FUNCTION_BLOCK FB_MotorControl
VAR_INPUT
	AxisRef 	:	AXIS_REF;
	//Position
	//Ready
	//Reset
	
END_VAR
VAR_OUTPUT
		error	: BOOL;
END_VAR

(*Internals*)
VAR
	(* Properties *)
	Enabled : BOOL := FALSE;	


	eInitMotor : (START, IN_PROCESS, DONE, ERROR);	
	eMoveABS : (START, IN_PROCESS, DONE, ERROR);

	//stMC_Reset : ST_MC_Reset;
	

	stSA_Reset	:   ST_MC_Status;
	
	
	
	fbMcPower	:	MC_POWER;
	fbMcHome	: 	MC_HOME;
	fbMcJog		:	MC_JOG;
	
	// Global
	bError 		: BOOL	; // := TRUE;
	nErrorID 	: LINT	; //Check type
	
	//Reset
	fbMcReset	:	MC_RESET;
	fbTriggerReset : R_TRIG;
	bResetDone : BOOL := FALSE;
	
	
	
	fbMoveVelocity	: MC_MoveVelocity;
	fbMoveRelative	: MC_MoveRelative;
	fbMoveAbsolute	: MC_MoveAbsolute;
	
	fbHalt	: MC_Halt;
	fbStop	: MC_Stop;
	
	fbSA_GetPosition : MC_ReadActualPosition;
	
	//Input: Command
	bCmdResetExe			:	BOOL	;
	bCmdPowerEnable			:	BOOL	;
	bCmdPowerEnablePositive	:	BOOL	;
	bCmdPowerEnableNegative	:	BOOL	;
	bCmdHomeExecute			:	BOOL	;
	bSA_HomeCamInput	:	BOOL	;
	
	bSA_JogFwd			:	BOOL	;
	bSA_JogRev			:	BOOL	;
	
	bSA_HaltExe			: 	BOOL	;
	bSA_StopExe			: 	BOOL	;
	
	//stStatusMoveVelocity	: ST_MC_CMD	;
	stSA_VelCmd1	: ST_MC_CMD;
	stSA_RelCmd1			: ST_MC_CMD	;
	stSA_AbsCmd1			: ST_MC_CMD	;
	
	//Variables / Parameters
	lrSA_PowerOverride	: LREAL;
	lrSA_HomePosition	: LREAL;
	lrSA_SetPosition	: LREAL;
	lrSA_JogVelocity	: LREAL;
	
	//Status
	//stSA_Reset			: ST_MC_Status;
	stSA_Power			: ST_MC_Status;
	stSA_Home			: ST_MC_Status;
	stSA_SetPosition	: ST_MC_Status;
	stSA_Jog			: ST_MC_Status;
	stSA_GetPosition	: ST_MC_Status;
	
	
	stSA_VelSts1		: ST_MC_Status;
	stSA_MoveRelative		: ST_MC_Status;
	stSA_AbsSts1		: ST_MC_Status;
	
	stSA_Halt			: ST_MC_Status;
	stSA_Stop			: ST_MC_Status;

END_VAR

AxisRef.ReadStatus();
GetStatus();
//Here the state machine needs to be processed or farmed out.



//For a move

//Has position changed from the current target.....






//This should be removed as seperate methods are added.
ExecuteCommands();

PROPERTY bStateEnable : BOOL
GET
bStateEnable := Enabled ;
END_GET
SET
Enabled := bStateEnable;
END_SET
END_PROPERTY

METHOD PRIVATE Enable : BOOL
VAR_INPUT
END_VAR
END_METHOD

METHOD PRIVATE ExecuteCommands : BOOL
VAR_INPUT
END_VAR

VAR
END_VAR
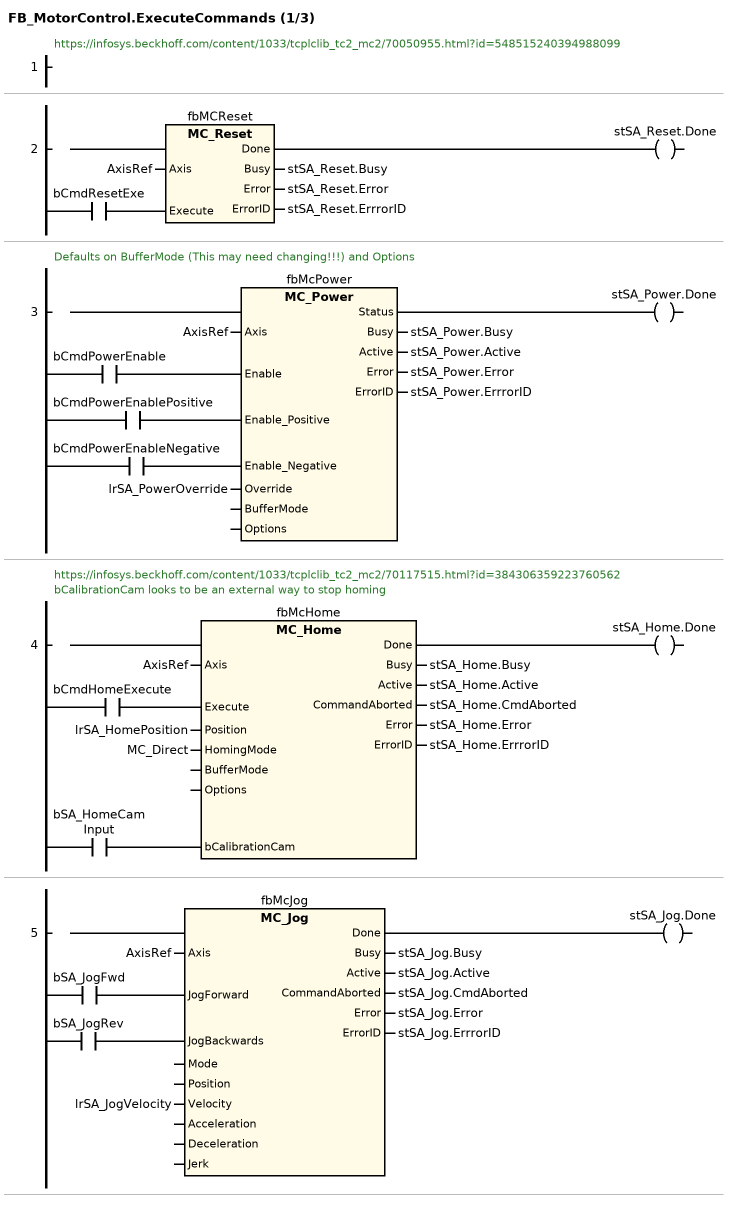
// NETWORK 1
// https://infosys.beckhoff.com/content/1033/tcplclib_tc2_mc2/70050955.html?id=548515240394988099

// NETWORK 2
fbMCReset(
    Axis := AxisRef,
    Execute := bCmdResetExe,
    Busy => stSA_Reset.Busy,
    Error => stSA_Reset.Error,
    ErrorID => stSA_Reset.ErrrorID); // MC_Reset
stSA_Reset.Done := fbMCReset.Done;

// NETWORK 3
// Defaults on BufferMode (This may need changing!!!) and Options
fbMcPower(
    Axis := AxisRef,
    Enable := bCmdPowerEnable,
    Enable_Positive := bCmdPowerEnablePositive,
    Enable_Negative := bCmdPowerEnableNegative,
    Override := lrSA_PowerOverride,
    Busy => stSA_Power.Busy,
    Active => stSA_Power.Active,
    Error => stSA_Power.Error,
    ErrorID => stSA_Power.ErrrorID); // MC_Power
stSA_Power.Done := fbMcPower.Status;

// NETWORK 4
// https://infosys.beckhoff.com/content/1033/tcplclib_tc2_mc2/70117515.html?id=384306359223760562
// bCalibrationCam looks to be an external way to stop homing
fbMcHome(
    Axis := AxisRef,
    Execute := bCmdHomeExecute,
    Position := lrSA_HomePosition,
    HomingMode := MC_Direct,
    bCalibrationCam := bSA_HomeCamInput,
    Busy => stSA_Home.Busy,
    Active => stSA_Home.Active,
    CommandAborted => stSA_Home.CmdAborted,
    Error => stSA_Home.Error,
    ErrorID => stSA_Home.ErrrorID); // MC_Home
stSA_Home.Done := fbMcHome.Done;

// NETWORK 5
fbMcJog(
    Axis := AxisRef,
    JogForward := bSA_JogFwd,
    JogBackwards := bSA_JogRev,
    Velocity := lrSA_JogVelocity,
    Busy => stSA_Jog.Busy,
    Active => stSA_Jog.Active,
    CommandAborted => stSA_Jog.CmdAborted,
    Error => stSA_Jog.Error,
    ErrorID => stSA_Jog.ErrrorID); // MC_Jog
stSA_Jog.Done := fbMcJog.Done;

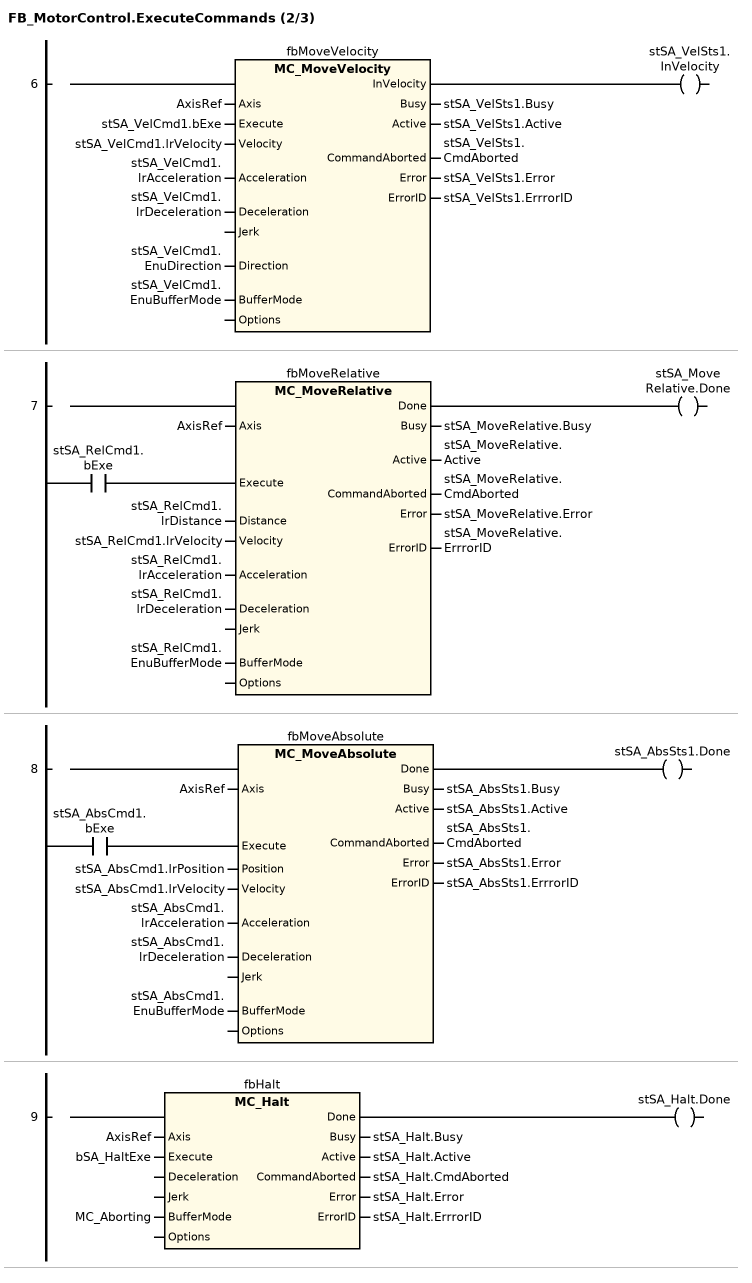
// NETWORK 6
fbMoveVelocity(
    Axis := AxisRef,
    Execute := stSA_VelCmd1.bExe,
    Velocity := stSA_VelCmd1.lrVelocity,
    Acceleration := stSA_VelCmd1.lrAcceleration,
    Deceleration := stSA_VelCmd1.lrDeceleration,
    Direction := stSA_VelCmd1.EnuDirection,
    BufferMode := stSA_VelCmd1.EnuBufferMode,
    Busy => stSA_VelSts1.Busy,
    Active => stSA_VelSts1.Active,
    CommandAborted => stSA_VelSts1.CmdAborted,
    Error => stSA_VelSts1.Error,
    ErrorID => stSA_VelSts1.ErrrorID); // MC_MoveVelocity
stSA_VelSts1.InVelocity := fbMoveVelocity.InVelocity;

// NETWORK 7
fbMoveRelative(
    Axis := AxisRef,
    Execute := stSA_RelCmd1.bExe,
    Distance := stSA_RelCmd1.lrDistance,
    Velocity := stSA_RelCmd1.lrVelocity,
    Acceleration := stSA_RelCmd1.lrAcceleration,
    Deceleration := stSA_RelCmd1.lrDeceleration,
    BufferMode := stSA_RelCmd1.EnuBufferMode,
    Busy => stSA_MoveRelative.Busy,
    Active => stSA_MoveRelative.Active,
    CommandAborted => stSA_MoveRelative.CmdAborted,
    Error => stSA_MoveRelative.Error,
    ErrorID => stSA_MoveRelative.ErrrorID); // MC_MoveRelative
stSA_MoveRelative.Done := fbMoveRelative.Done;

// NETWORK 8
fbMoveAbsolute(
    Axis := AxisRef,
    Execute := stSA_AbsCmd1.bExe,
    Position := stSA_AbsCmd1.lrPosition,
    Velocity := stSA_AbsCmd1.lrVelocity,
    Acceleration := stSA_AbsCmd1.lrAcceleration,
    Deceleration := stSA_AbsCmd1.lrDeceleration,
    BufferMode := stSA_AbsCmd1.EnuBufferMode,
    Busy => stSA_AbsSts1.Busy,
    Active => stSA_AbsSts1.Active,
    CommandAborted => stSA_AbsSts1.CmdAborted,
    Error => stSA_AbsSts1.Error,
    ErrorID => stSA_AbsSts1.ErrrorID); // MC_MoveAbsolute
stSA_AbsSts1.Done := fbMoveAbsolute.Done;

// NETWORK 9
fbHalt(
    Axis := AxisRef,
    Execute := bSA_HaltExe,
    BufferMode := MC_Aborting,
    Busy => stSA_Halt.Busy,
    Active => stSA_Halt.Active,
    CommandAborted => stSA_Halt.CmdAborted,
    Error => stSA_Halt.Error,
    ErrorID => stSA_Halt.ErrrorID); // MC_Halt
stSA_Halt.Done := fbHalt.Done;

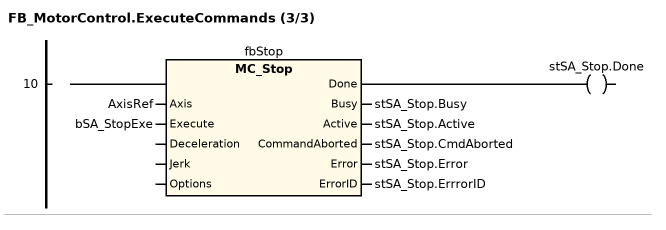
// NETWORK 10
fbStop(
    Axis := AxisRef,
    Execute := bSA_StopExe,
    Busy => stSA_Stop.Busy,
    Active => stSA_Stop.Active,
    CommandAborted => stSA_Stop.CmdAborted,
    Error => stSA_Stop.Error,
    ErrorID => stSA_Stop.ErrrorID); // MC_Stop
stSA_Stop.Done := fbStop.Done;
END_METHOD

METHOD PRIVATE GetStatus : BOOL
VAR_INPUT
END_VAR
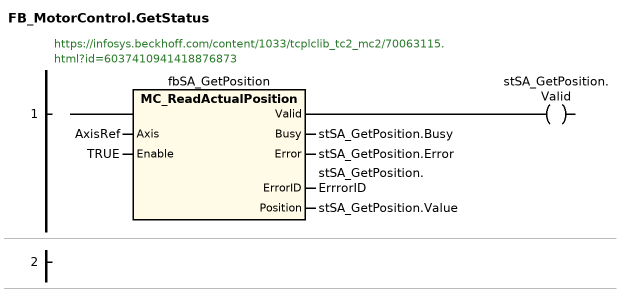
// NETWORK 1
// https://infosys.beckhoff.com/content/1033/tcplclib_tc2_mc2/70063115.html?id=6037410941418876873
fbSA_GetPosition(
    Axis := AxisRef,
    Enable := TRUE,
    Busy => stSA_GetPosition.Busy,
    Error => stSA_GetPosition.Error,
    ErrorID => stSA_GetPosition.ErrrorID,
    Position => stSA_GetPosition.Value); // MC_ReadActualPosition
stSA_GetPosition.Valid := fbSA_GetPosition.Valid;

// NETWORK 2
END_METHOD

METHOD Halt : BOOL
VAR_INPUT
END_VAR
END_METHOD

METHOD PUBLIC MoveAbs : BOOL
VAR_INPUT
	Distance 		: LREAL;
	Velocity 		: LREAL;

//https://infosys.beckhoff.com/content/1033/tcplclib_tc2_mc2/70147595.html?id=4401319670753010232
	mcBufferMode	: MC_BufferMode;
(*  MC_Aborting,			Cancels P1 and  moves to P2
    MC_Buffered,			Moves to P1, stops and moves to P2
    MC_BlendingLow, MC_BlendingPrevious, MC_BlendingNext, MC_BlendingHigh	Change the way speed is blended  BlendingLow would generaly be the one I'd choose. *)
	
END_VAR
VAR
	

END_VAR
(*  It is not needed to wait for the end of a move, will be qued - but do need to ensure Execute operates with a rising edge.
	Not concerned about "loosing" commands, no buffer needed, only the last command matters.*)   

(*
If in Error state ignore.

If "Busy"	Execute == FALSE;

if Execute == FALSE can send new command

*)	

	
	
//CASE fbMoveAbsolute.Execute OF
//	TRUE: 
	
//	IN_PROCESS:

//	DONE:
	
	
//END_CASE

//Does this have meaning.....
MoveAbs := TRUE;
END_METHOD

METHOD Reset : BOOL
VAR_INPUT
	bDriveReset : Bool;
END_VAR
// Indicate that the Reset is in progress
IF NOT bDriveReset THEN
	bResetDone := FALSE;
END_IF

// Trigger
fbTriggerReset(CLK := bDriveReset);

IF fbTriggerReset.Q THEN
	//Is this meant to be sending a halt to the motor at the same time....?
	//If so why not as a command - seems more of a status....
	
	//bHaltDone := FALSE;
	fbMcReset(Execute := TRUE, Axis := AxisRef);
ELSE				
	fbMcReset(Axis := AxisRef); //What happens to the unchanged values - defaults......TEST?
END_IF;
 
// Done / Error 
IF fbMcReset.Done OR fbMcReset.Error THEN
	bError := fbMcReset.Error;
	nErrorID := fbMcReset.ErrorID;
	bResetDone := fbMcReset.Done;
	
	fbMcReset(Execute := FALSE, Axis := AxisRef);
END_IF
END_METHOD

METHOD Stop : BOOL
VAR_INPUT
END_VAR
END_METHOD

END_FUNCTION_BLOCK

(* stored: Version 1.1.0.1, ProductVersion 3.1.4024.11
   POU FB_MotorControl: Id {9b26cca3-dfb1-468b-828a-5d52f957fd6b}, SpecialFunc None
   Property bStateEnable: Id {33d52600-d274-4031-889c-2e201010dccb}
   Get Get: Id {7ef59478-eeec-47f5-985d-805d6da9dde0}
   Set Set: Id {11f65afe-6c13-496b-bfdd-5fd891f1923d}
   Method Enable: Id {3d9238b1-74ad-4672-b4ef-014884ddfba6}
   Method ExecuteCommands: Id {489d89ce-c8ae-4ad4-85e5-887c50bac62e}
   Method GetStatus: Id {17d03984-c95a-4c5d-b9a7-5c1d935ee030}
   Method Halt: Id {e714a366-01da-41dc-a0ee-ef934f68efa7}
   Method MoveAbs: Id {66624a6b-dded-4da6-b083-e23604a33508}
   Method Reset: Id {db5a6dee-a30a-4d6d-a1e0-2dd4b7425fc5}
   Method Stop: Id {bf57bcbf-4a9d-498b-aa4c-b637e7f4fe66} *)
